// TIA Portal V19 export
FUNCTION_BLOCK "FB_FU_OUT_TW"   // FB12, LAD
TITLE = Ausgabe Einzel-FU
{ S7_Optimized_Access := 'TRUE' }
// stored: AutoNumber false, IsIECCheckEnabled true, MemoryReserve 100, SetENOAutomatically false
   VAR_INPUT
      Req_High : Bool;   // Anforderung Vorwärts/Heben
      Req_Low : Bool;   // Anforderun Rückwärts/Senken
   END_VAR
   VAR_IN_OUT
      Reglersperre : Bool;
      Freigabe_Stopp : Bool;
      Freigabe_Halt : Bool;
      Break_ok : Bool;
      SollSpeed : Int;   // Geschwindigkeit Fahren in %
      Ist_Speed : Int;
      PAW_Speed : Int;
      PEW_Speed : Int;
   END_VAR
   VAR RETAIN
      maxSpeed : Real := 7500.0;   // maximale Ausgabe (entspricht 100%)
      Faktor { ExternalAccessible := 'False'; ExternalVisible := 'False'; ExternalWritable := 'False'} : Real := 100.0;
      minSpeed : Int := 750;   // Freigabe nehmen unterhalb diesen Wertes im PEW
   END_VAR
   VAR_TEMP
      TempSpeed : Real;
      Faktor_Sim : Real;
      Delta : Int;
   END_VAR
BEGIN

REGION Network 1 (SCL): Istwert erfassen
   REGION Istwert erfassen
       // Statement section REGION
       #Ist_Speed:=REAL_TO_INT((INT_TO_REAL(#PEW_Speed)/#maxSpeed) * #Faktor);
   END_REGION
END_REGION

REGION Network 2 (SCL): Ausgabe Speed
   REGION Ausgabe Speed

       //Not-Halt --> sofort aus
       IF "DB_ANLAGE".BA.Not_Aus THEN
           #Reglersperre := TRUE;
           #Freigabe_Stopp := FALSE;
           #PAW_Speed := 0;

           //vorwärts/hoch positive Ausgabe    
       ELSIF #Req_High AND #SollSpeed <> 0 THEN
           #Reglersperre := FALSE;
           #Freigabe_Stopp := TRUE;
           #PAW_Speed := REAL_TO_INT(INT_TO_REAL(#SollSpeed) / #Faktor * #maxSpeed);

           //rückwärts/runter negative Ausgabe    
       ELSIF #Req_Low AND #SollSpeed <> 0 THEN
           #Reglersperre := FALSE;
           #Freigabe_Stopp := TRUE;
           #PAW_Speed := REAL_TO_INT(INT_TO_REAL(#SollSpeed) / #Faktor * #maxSpeed * -1.0);

           //sonst aus    
       ELSE
           #Freigabe_Stopp := #PEW_Speed >= #minSpeed;
           #Reglersperre := FALSE;
           #PAW_Speed := 0;
       END_IF;

       #Freigabe_Halt := #Freigabe_Stopp;
       #Break_ok := NOT #Freigabe_Stopp AND #Ist_Speed=0;

   END_REGION
END_REGION

REGION Network 3 (SCL): Simulation
   REGION Simulation

       IF "DB_ANLAGE".BA.Simulation THEN

           //Abfahrrampe berechnen
           #Faktor_Sim := 15.0; //500ms von 7500 auf 0 (7500.0/500.0)
           //Korrekturwert berechnen
           #Delta := REAL_TO_INT(#Faktor_Sim * INT_TO_REAL("DI_FW_MANAGER".akt_CT));

           //Geschwindigkeit reduzieren
           IF #PEW_Speed > #PAW_Speed THEN
               #PEW_Speed := #PEW_Speed - #Delta;
               IF #PEW_Speed <= #PAW_Speed THEN
                   #PEW_Speed := #PAW_Speed;
               END_IF;

               //Geschwindigkeit erhöhen
           ELSIF #PEW_Speed < #PAW_Speed THEN
               #PEW_Speed := #PEW_Speed + #Delta;
               IF #PEW_Speed >= #PAW_Speed THEN
                   #PEW_Speed := #PAW_Speed;
               END_IF;

           ELSE
               #PEW_Speed := #PAW_Speed;
           END_IF; 

       END_IF;
   END_REGION
END_REGION
END_FUNCTION_BLOCK
